(*
SPDX-FileCopyrightText: © 2026 Oleksandr Tiutyk <trofimich@gmail.com>
SPDX-License-Identifier: MIT
License: https://opensource.org/license/mit
*)

(*!
<summary>Writes messages and exception diagnostics to the ADS log.</summary>
<description>
Use this backend for short diagnostics in the standard ADS log. LogManager provides a separate instance for
each cyclic task. Requires no cyclic work. Direct concurrent use has no established guarantee in this
contract: formatting uses call-local storage, but that alone does not establish concurrency guarantees for
ADSLOGSTR and all nested calls. This is not a confirmed concurrency defect. For a single-task backend access path from multiple sending
tasks, use the QueuedLogger wrapper from the Loggers library and do not call the backend concurrently outside
that wrapper. This backend is intended for short diagnostics. Each TryLogMessage call emits one ADS record;
text exceeding the conversion or ADS output capacity is truncated at the end, without splitting it into
multiple records. The optional number prefix consumes part of that capacity. Message text is passed as the ADS
string argument with a fixed format, so format tokens in the message remain literal text. Exception logging
accepts IReadOnlyException and reads borrowed diagnostics without transferring ownership. Implementations must
not retain exception references beyond their task cleanup. TryLog methods must satisfy the no-throw contract
even when called directly, without LogManager. Does not propagate exceptions, including failures while reading
or formatting diagnostics and calling the backend; returns FALSE instead. Already emitted entries are not
rolled back, so FALSE may follow partial output. Caught exceptions are not logged again. The fatal allocation
latch is preserved for RaiseIfAllocationFailed at the task boundary outside recoverable handlers.
</description>
*)

{attribute 'no_explicit_call' := 'do not call this function block directly'}
FUNCTION_BLOCK AdsLogger EXTENDS Object IMPLEMENTS ILogger
VAR_STAT
	//! <summary>Class name shared by all instances of this function block.</summary>
	{attribute 'hide'} 
	_ClassName : STRING := __POUNAME();
END_VAR

{attribute 'monitoring' := 'call'}
PROPERTY ClassName : REFERENCE TO STRING
GET
ClassName REF= _ClassName;
END_GET
END_PROPERTY

(*!
<summary>Completes without work because this logger has no cyclic processing.</summary>
<description>Does not raise exceptions.</description>
*)
METHOD Execute
// nothing to do for ADS logger
END_METHOD

(*!
<summary>Provides the library namespace used in diagnostics.</summary>
<description>
Borrowed read-only reference to the compiler-initialized library namespace; no ownership transfer.
</description>
*)
{attribute 'monitoring' := 'call'}
PROPERTY NamespaceName : REFERENCE TO STRING
GET
NamespaceName REF= CurrentNamespace.Name;
END_GET
END_PROPERTY

(*!
<summary>Reports the byte size of this concrete instance.</summary>
<description>
Uses XSIZEOF on the instance. Does not include separately allocated payloads or prove that an arbitrary
address is valid.
</description>
*)
{attribute 'monitoring' := 'call'}
PROPERTY SelfSize : ULINT
GET
SelfSize := XSIZEOF(THIS^);
END_GET
END_PROPERTY

(*!
<summary>Attempts to log a borrowed error without propagating exceptions.</summary>
<description>
Borrows inputs only for the call. TRUE reports backend acceptance, not guaranteed durable storage. Does not
propagate exceptions, including failures while reading or formatting diagnostics and calling the backend;
returns FALSE instead. Already emitted entries are not rolled back, so FALSE may follow partial output. Caught
exceptions are not logged again. The fatal allocation latch is preserved for RaiseIfAllocationFailed at the
task boundary outside recoverable handlers. Descendants cannot replace this non-throwing ADS logging path;
implement ILogger separately for another backend.
Returns FALSE when fatal allocation state is observed before work or after nested calls. The latch remains
set for the caller's task boundary; already accepted or emitted records are not rolled back.
</description>
*)
METHOD FINAL TryLogError : BOOL
VAR_INPUT
	error : REFERENCE TO ERROR;
	messageNumber : REFERENCE TO ULINT := 0;
END_VAR
VAR
	message : ERROR_MESSAGE;
END_VAR
__TRY
	IF DynamicMemoryManager.HasAllocationFailed OR_ELSE NOT __ISVALIDREF(error) THEN
		RETURN;
	END_IF

	message := error.ToString(
		sourceDisplayMode := ERROR_SOURCE_DISPLAY_MODE.TOP_AND_ROOT,
		timestampDisplayMode := TIMESTAMP_DISPLAY_MODE.LOCAL
	);

	TryLogError := TryLogMessage(
		category := SEL(error.Severity = ERROR_SEVERITY.CRITICAL, LOG_CATEGORY.ERROR, LOG_CATEGORY.CRITICAL_ERROR),
		message := message,
		messageNumber := messageNumber
	);

	IF DynamicMemoryManager.HasAllocationFailed THEN
		TryLogError := FALSE;
	END_IF
__CATCH
	TryLogError := FALSE;
__ENDTRY
END_METHOD

(*!
<summary>Attempts to log diagnostic information from a read-only exception view.</summary>
<description>
Borrows the exception for the call without clearing it or taking ownership. The exception and its inner causes
must remain live while their diagnostics are read. Logging does not extend their lifetime. Does not propagate
exceptions, including failures while reading or formatting diagnostics and calling the backend; returns FALSE
instead. Already emitted entries are not rolled back, so FALSE may follow partial output. Caught exceptions
are not logged again. The fatal allocation latch is preserved for RaiseIfAllocationFailed at the task boundary
outside recoverable handlers. Descendants cannot replace this non-throwing ADS logging path; implement ILogger
separately for another backend.
Returns FALSE when fatal allocation state is observed before work or after nested calls. The latch remains
set for the caller's task boundary; already accepted or emitted records are not rolled back.
</description>
<param name="exception">Exception view to read; null is ignored.</param>
<param name="severity">Severity used to select the log category.</param>
<param name="messageNumber">
Optional number forwarded to the ordinary or single-cause message, or to the header of a multi-cause
aggregate.
</param>
*)
METHOD FINAL TryLogException : BOOL
VAR_INPUT
	exception : IReadOnlyException;
	severity : ERROR_SEVERITY;
	messageNumber : REFERENCE TO ULINT := 0;
END_VAR
VAR
	message : ERROR_MESSAGE;
	aggregateException : IAggregateException;
	innerExceptionCount : UINT;
	innerException : IReadOnlyException;
	i : DINT;
END_VAR
__TRY
	IF DynamicMemoryManager.HasAllocationFailed OR_ELSE exception = 0 THEN
		RETURN;
	END_IF

	IF __QUERYINTERFACE(exception, aggregateException) THEN
		innerExceptionCount := aggregateException.InnerExceptionCount;
	END_IF

	IF innerExceptionCount = 0 THEN
		message := exception.GetMessage(showSource := TRUE, timestampDisplayMode := TIMESTAMP_DISPLAY_MODE.LOCAL);

		TryLogException := TryLogMessage(
			category := SEL(severity = ERROR_SEVERITY.CRITICAL, LOG_CATEGORY.ERROR, LOG_CATEGORY.CRITICAL_ERROR),
			message := message,
			messageNumber := messageNumber
		);
	ELSE
		IF innerExceptionCount > 1 THEN
			// reverce order
			TryLogException := TryLogMessage(category := LOG_CATEGORY.ERROR, message := "<<< aggregate exception end <<<");

			FOR i := TO_DINT(innerExceptionCount) - 1 TO 0 BY -1 DO
				innerException := aggregateException.GetInnerException(index := i);

				IF DynamicMemoryManager.HasAllocationFailed THEN
					TryLogException := FALSE;
					RETURN;
				END_IF

				message := WideStrings.Concat255(
					"  ",
					innerException.GetMessage(showSource := TRUE, timestampDisplayMode := TIMESTAMP_DISPLAY_MODE.LOCAL)
				);

				TryLogException := TryLogException AND TryLogMessage(
					category := SEL(severity = ERROR_SEVERITY.CRITICAL, LOG_CATEGORY.ERROR, LOG_CATEGORY.CRITICAL_ERROR),
					message := message
				);

				IF DynamicMemoryManager.HasAllocationFailed THEN
					TryLogException := FALSE;
					RETURN;
				END_IF
			END_FOR

			TryLogException := TryLogException AND TryLogMessage(
				category := SEL(severity = ERROR_SEVERITY.CRITICAL, LOG_CATEGORY.ERROR, LOG_CATEGORY.CRITICAL_ERROR),
				message := ">>> aggregate exception start >>>",
				messageNumber := messageNumber
			);
		ELSE
			innerException := aggregateException.GetInnerException(index := 0);

			IF DynamicMemoryManager.HasAllocationFailed THEN
				TryLogException := FALSE;
				RETURN;
			END_IF

			message := innerException.GetMessage(showSource := TRUE, timestampDisplayMode := TIMESTAMP_DISPLAY_MODE.LOCAL);

			TryLogException := TryLogMessage(
				category := SEL(severity = ERROR_SEVERITY.CRITICAL, LOG_CATEGORY.ERROR, LOG_CATEGORY.CRITICAL_ERROR),
				message := message,
				messageNumber := messageNumber
			);
		END_IF
	END_IF

	IF DynamicMemoryManager.HasAllocationFailed THEN
		TryLogException := FALSE;
	END_IF
__CATCH
	TryLogException := FALSE;
__ENDTRY
END_METHOD

(*!
<summary>Attempts to write message text and an optional message number to the ADS log.</summary>
<description>
Requests log output for every severity (hint, warning or error). Uses the fixed ADS format %s and passes the
converted text as its string argument. Format tokens within the message remain literal. Bounds the converted
text, including any number prefix, to 253 bytes before calling ADSLOGSTR. Emits one record with no continuation records. Borrows arguments only for the call.
Returns TRUE when ADSLOGSTR returns success; the entire original ERROR_MESSAGE may not fit in the ADS output.
Does not propagate exceptions,
including failures while reading or formatting diagnostics and calling the backend; returns FALSE instead.
Already emitted entries are not rolled back, so FALSE may follow partial output. Caught exceptions are not
logged again. The fatal allocation latch is preserved for RaiseIfAllocationFailed at the task boundary outside
recoverable handlers. Descendants cannot replace this non-throwing ADS logging path; implement ILogger
separately for another backend.
Returns FALSE when fatal allocation state is observed before work or after nested calls. The latch remains
set for the caller's task boundary; already accepted or emitted records are not rolled back.
</description>
<param name="category">Category used to select the ADS message mask and optional number prefix.</param>
<param name="message">Message text converted to STRING for ADS output.</param>
<param name="messageNumber">Optional borrowed number prepended to the message.</param>
*)
METHOD FINAL TryLogMessage : BOOL
VAR_INPUT
	category : LOG_CATEGORY;	
END_VAR
VAR_IN_OUT CONSTANT
	message : ERROR_MESSAGE;
END_VAR
VAR_INPUT
	messageNumber : REFERENCE TO ULINT := 0;
END_VAR
VAR
	messageControlMask : DWORD;
	adsText : STRING(253); // ADSLOGSTR limits the formatted message to 253 bytes.
END_VAR
__TRY
	IF DynamicMemoryManager.HasAllocationFailed THEN
		RETURN;
	END_IF

	CASE category OF
		LOG_CATEGORY.DEBUG, LOG_CATEGORY.INFORMATION:
			messageControlMask := Tc2_System.Global_Variables.ADSLOG_MSGTYPE_HINT
				OR Tc2_System.Global_Variables.ADSLOG_MSGTYPE_LOG;

		LOG_CATEGORY.WARNING:
			messageControlMask := Tc2_System.Global_Variables.ADSLOG_MSGTYPE_WARN
				OR Tc2_System.Global_Variables.ADSLOG_MSGTYPE_LOG;

		LOG_CATEGORY.ERROR, LOG_CATEGORY.CRITICAL_ERROR:
			messageControlMask := Tc2_System.Global_Variables.ADSLOG_MSGTYPE_ERROR
				OR Tc2_System.Global_Variables.ADSLOG_MSGTYPE_LOG;
	END_CASE

	IF __ISVALIDREF(messageNumber) THEN
		adsText := Strings.Concat255(
			TO_STRING(Exceptions.MESSAGE_NUMBER_PREFIX),
			Exceptions.LOG_CATEGORY_PREFIXES[category],
			TO_STRING(messageNumber),
			TO_STRING(Exceptions.MESSAGE_NUMBER_SUFFIX),
			TO_STRING(message)
		);
	ELSE
		adsText := TO_STRING(message);
	END_IF

	TryLogMessage := Tc2_System.ADSLOGSTR(
		msgCtrlMask := messageControlMask,
		msgFmtStr := '%s',
		strArg := adsText
	) = 0;

	IF DynamicMemoryManager.HasAllocationFailed THEN
		TryLogMessage := FALSE;
	END_IF
__CATCH
	TryLogMessage := FALSE;
__ENDTRY
END_METHOD

END_FUNCTION_BLOCK

(* stored: Version 1.1.0.1
   POU AdsLogger: Id {c95de8ac-0505-4250-b81e-2b0cbe2bb2ed}, SpecialFunc None
   Property ClassName: Id {c900fbb9-86d0-4a3f-9595-f30e1df1d1f1}
   Get Get: Id {910140d1-6146-4f27-82a4-105ab45c7077}
   Method Execute: Id {7f679376-d6c2-4628-9f18-706629e6a200}
   Property NamespaceName: Id {c38469fc-4ff8-41a9-b499-75e413a00bb3}
   Get Get: Id {bcccda69-31bf-4d44-868c-2415428102e1}
   Property SelfSize: Id {c266c68f-d111-413c-997b-ce427475c7b9}
   Get Get: Id {368ffd0e-de98-47d3-99fe-4d83a0af5f22}
   Method TryLogError: Id {20bf6186-2dc6-4029-8680-18c8f237e377}
   Method TryLogException: Id {52444f42-e6c7-4828-baa7-3f12fe45268b}
   Method TryLogMessage: Id {936430cf-8fdd-47d1-875f-690550891879} *)
